// TIA Portal V19 export
FUNCTION "ALARMS" : Void   // FC10, LAD
{ S7_Optimized_Access := 'TRUE' }
// stored: SetENOAutomatically false
   VAR_TEMP   // added for the SCL form of the ladder/FBD networks
      _w1 : Bool;
   END_VAR
BEGIN

REGION Network 1: ERROR BIT
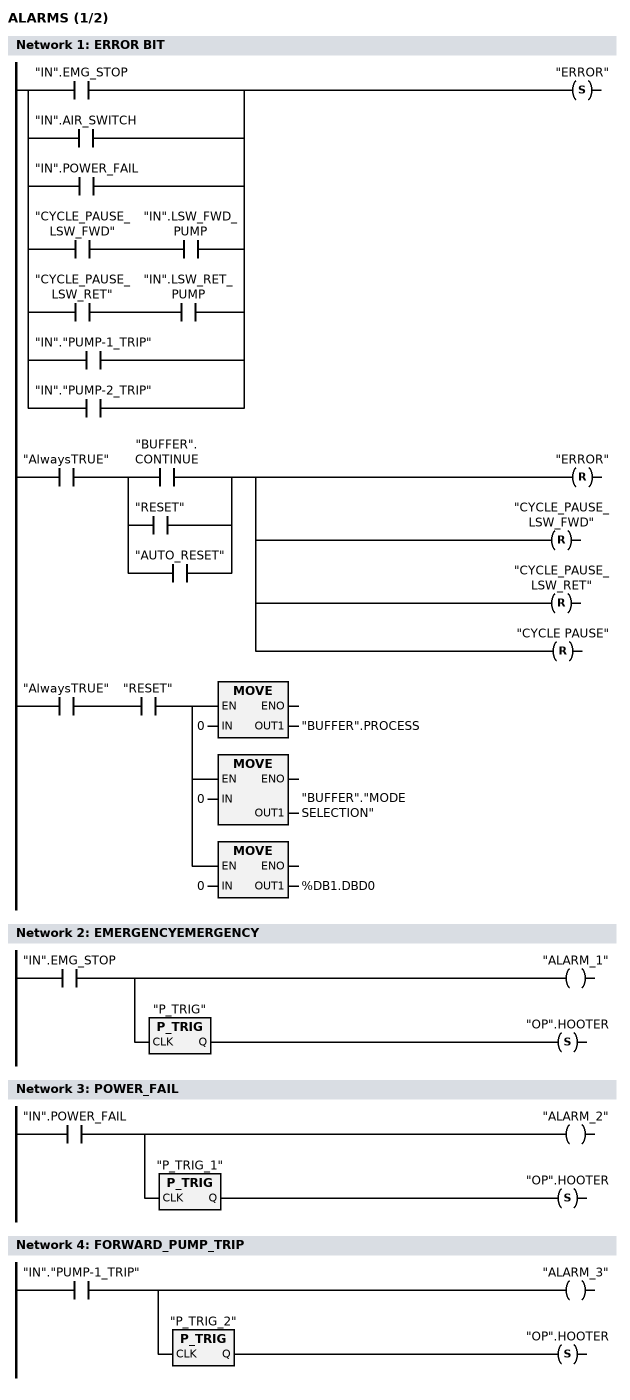
   RUNG wire#powerrail
      Contact( "IN".EMG_STOP )
      wire#w1
      S_Coil( "ERROR" )
   END_RUNG
   RUNG wire#powerrail
      Contact( "IN".AIR_SWITCH )
   END_RUNG wire#w1
   RUNG wire#powerrail
      Contact( "IN".POWER_FAIL )
   END_RUNG wire#w1
   RUNG wire#powerrail
      Contact( "CYCLE_PAUSE_LSW_FWD" )
      Contact( "IN".LSW_FWD_PUMP )
   END_RUNG wire#w1
   RUNG wire#powerrail
      Contact( "CYCLE_PAUSE_LSW_RET" )
      Contact( "IN".LSW_RET_PUMP )
   END_RUNG wire#w1
   RUNG wire#powerrail
      Contact( "IN"."PUMP-1_TRIP" )
   END_RUNG wire#w1
   RUNG wire#powerrail
      Contact( "IN"."PUMP-2_TRIP" )
   END_RUNG wire#w1
   RUNG wire#powerrail
      Contact( "AlwaysTRUE" )
      wire#w2
      Contact( "BUFFER".CONTINUE )
      wire#w3
      R_Coil( "ERROR" )
   END_RUNG
   RUNG wire#w2
      Contact( "RESET" )
   END_RUNG wire#w3
   RUNG wire#w2
      Contact( "AUTO_RESET" )
   END_RUNG wire#w3
   RUNG wire#w3
      R_Coil( "CYCLE_PAUSE_LSW_FWD" )
   END_RUNG
   RUNG wire#w3
      R_Coil( "CYCLE_PAUSE_LSW_RET" )
   END_RUNG
   RUNG wire#w3
      R_Coil( "CYCLE PAUSE" )
   END_RUNG
   RUNG wire#powerrail
      Contact( "AlwaysTRUE" )
      Contact( "RESET" )
      wire#w4
      Move(in := 0, out1 => "BUFFER".PROCESS)
   END_RUNG
   RUNG wire#w4
      Move(in := 0, out1 => "BUFFER"."MODE SELECTION")
   END_RUNG
   RUNG wire#w4
      Move(in := 0, out1 => %DB1.DBD0)
   END_RUNG
   // the same network as SCL:
   IF "IN".EMG_STOP OR "IN".AIR_SWITCH OR "IN".POWER_FAIL OR ("CYCLE_PAUSE_LSW_FWD" AND "IN".LSW_FWD_PUMP) OR ("CYCLE_PAUSE_LSW_RET" AND "IN".LSW_RET_PUMP) OR "IN"."PUMP-1_TRIP" OR "IN"."PUMP-2_TRIP" THEN
       "ERROR" := TRUE;
   END_IF;
   IF "AlwaysTRUE" AND ("BUFFER".CONTINUE OR "RESET" OR "AUTO_RESET") THEN
       "ERROR" := FALSE;
       "CYCLE_PAUSE_LSW_FWD" := FALSE;
       "CYCLE_PAUSE_LSW_RET" := FALSE;
       "CYCLE PAUSE" := FALSE;
   END_IF;
   IF "AlwaysTRUE" AND "RESET" THEN
       "BUFFER".PROCESS := 0;
       "BUFFER"."MODE SELECTION" := 0;
       %DB1.DBD0 := 0;
   END_IF;
END_REGION

REGION Network 2: EMERGENCYEMERGENCY
   RUNG wire#powerrail
      Contact( "IN".EMG_STOP )
      wire#w1
      Coil( "ALARM_1" )
   END_RUNG
   RUNG wire#w1
      P_Trig( "P_TRIG" )
      S_Coil( "OP".HOOTER )
   END_RUNG
   // the same network as SCL:
   "ALARM_1" := "IN".EMG_STOP;
   #_w1 := "IN".EMG_STOP AND NOT "P_TRIG";   // rising edge
   "P_TRIG" := "IN".EMG_STOP;
   IF #_w1 THEN "OP".HOOTER := TRUE; END_IF;
END_REGION

REGION Network 3: POWER_FAIL
   RUNG wire#powerrail
      Contact( "IN".POWER_FAIL )
      wire#w1
      Coil( "ALARM_2" )
   END_RUNG
   RUNG wire#w1
      P_Trig( "P_TRIG_1" )
      S_Coil( "OP".HOOTER )
   END_RUNG
   // the same network as SCL:
   "ALARM_2" := "IN".POWER_FAIL;
   #_w1 := "IN".POWER_FAIL AND NOT "P_TRIG_1";   // rising edge
   "P_TRIG_1" := "IN".POWER_FAIL;
   IF #_w1 THEN "OP".HOOTER := TRUE; END_IF;
END_REGION

REGION Network 4: FORWARD_PUMP_TRIP
   RUNG wire#powerrail
      Contact( "IN"."PUMP-1_TRIP" )
      wire#w1
      Coil( "ALARM_3" )
   END_RUNG
   RUNG wire#w1
      P_Trig( "P_TRIG_2" )
      S_Coil( "OP".HOOTER )
   END_RUNG
   // the same network as SCL:
   "ALARM_3" := "IN"."PUMP-1_TRIP";
   #_w1 := "IN"."PUMP-1_TRIP" AND NOT "P_TRIG_2";   // rising edge
   "P_TRIG_2" := "IN"."PUMP-1_TRIP";
   IF #_w1 THEN "OP".HOOTER := TRUE; END_IF;
END_REGION

REGION Network 5: RETURN_PUMP_TRIP
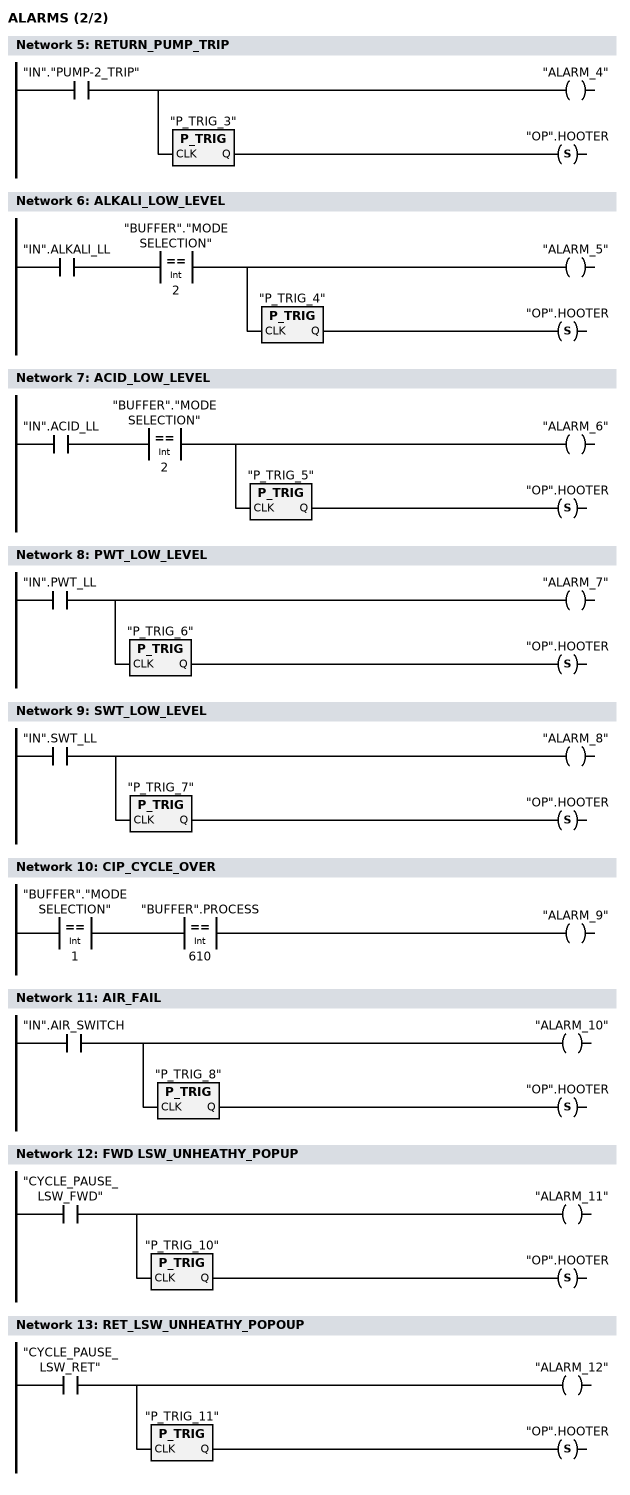
   RUNG wire#powerrail
      Contact( "IN"."PUMP-2_TRIP" )
      wire#w1
      Coil( "ALARM_4" )
   END_RUNG
   RUNG wire#w1
      P_Trig( "P_TRIG_3" )
      S_Coil( "OP".HOOTER )
   END_RUNG
   // the same network as SCL:
   "ALARM_4" := "IN"."PUMP-2_TRIP";
   #_w1 := "IN"."PUMP-2_TRIP" AND NOT "P_TRIG_3";   // rising edge
   "P_TRIG_3" := "IN"."PUMP-2_TRIP";
   IF #_w1 THEN "OP".HOOTER := TRUE; END_IF;
END_REGION

REGION Network 6: ALKALI_LOW_LEVEL
   RUNG wire#powerrail
      Contact( "IN".ALKALI_LL )
      { S7_Templates := "SrcType := Int" } EQ_Contact(in1 := "BUFFER"."MODE SELECTION", in2 := 2)
      wire#w1
      Coil( "ALARM_5" )
   END_RUNG
   RUNG wire#w1
      P_Trig( "P_TRIG_4" )
      S_Coil( "OP".HOOTER )
   END_RUNG
   // the same network as SCL:
   "ALARM_5" := "IN".ALKALI_LL AND ("BUFFER"."MODE SELECTION" = 2);
   #_w1 := "ALARM_5" AND NOT "P_TRIG_4";   // rising edge
   "P_TRIG_4" := "ALARM_5";
   IF #_w1 THEN "OP".HOOTER := TRUE; END_IF;
END_REGION

REGION Network 7: ACID_LOW_LEVEL
   RUNG wire#powerrail
      Contact( "IN".ACID_LL )
      { S7_Templates := "SrcType := Int" } EQ_Contact(in1 := "BUFFER"."MODE SELECTION", in2 := 2)
      wire#w1
      Coil( "ALARM_6" )
   END_RUNG
   RUNG wire#w1
      P_Trig( "P_TRIG_5" )
      S_Coil( "OP".HOOTER )
   END_RUNG
   // the same network as SCL:
   "ALARM_6" := "IN".ACID_LL AND ("BUFFER"."MODE SELECTION" = 2);
   #_w1 := "ALARM_6" AND NOT "P_TRIG_5";   // rising edge
   "P_TRIG_5" := "ALARM_6";
   IF #_w1 THEN "OP".HOOTER := TRUE; END_IF;
END_REGION

REGION Network 8: PWT_LOW_LEVEL
   RUNG wire#powerrail
      Contact( "IN".PWT_LL )
      wire#w1
      Coil( "ALARM_7" )
   END_RUNG
   RUNG wire#w1
      P_Trig( "P_TRIG_6" )
      S_Coil( "OP".HOOTER )
   END_RUNG
   // the same network as SCL:
   "ALARM_7" := "IN".PWT_LL;
   #_w1 := "IN".PWT_LL AND NOT "P_TRIG_6";   // rising edge
   "P_TRIG_6" := "IN".PWT_LL;
   IF #_w1 THEN "OP".HOOTER := TRUE; END_IF;
END_REGION

REGION Network 9: SWT_LOW_LEVEL
   RUNG wire#powerrail
      Contact( "IN".SWT_LL )
      wire#w1
      Coil( "ALARM_8" )
   END_RUNG
   RUNG wire#w1
      P_Trig( "P_TRIG_7" )
      S_Coil( "OP".HOOTER )
   END_RUNG
   // the same network as SCL:
   "ALARM_8" := "IN".SWT_LL;
   #_w1 := "IN".SWT_LL AND NOT "P_TRIG_7";   // rising edge
   "P_TRIG_7" := "IN".SWT_LL;
   IF #_w1 THEN "OP".HOOTER := TRUE; END_IF;
END_REGION

REGION Network 10: CIP_CYCLE_OVER
   RUNG wire#powerrail
      { S7_Templates := "SrcType := Int" } EQ_Contact(in1 := "BUFFER"."MODE SELECTION", in2 := 1)
      { S7_Templates := "SrcType := Int" } EQ_Contact(in1 := "BUFFER".PROCESS, in2 := 610)
      Coil( "ALARM_9" )
   END_RUNG
   // the same network as SCL:
   "ALARM_9" := ("BUFFER"."MODE SELECTION" = 1) AND ("BUFFER".PROCESS = 610);
END_REGION

REGION Network 11: AIR_FAIL
   RUNG wire#powerrail
      Contact( "IN".AIR_SWITCH )
      wire#w1
      Coil( "ALARM_10" )
   END_RUNG
   RUNG wire#w1
      P_Trig( "P_TRIG_8" )
      S_Coil( "OP".HOOTER )
   END_RUNG
   // the same network as SCL:
   "ALARM_10" := "IN".AIR_SWITCH;
   #_w1 := "IN".AIR_SWITCH AND NOT "P_TRIG_8";   // rising edge
   "P_TRIG_8" := "IN".AIR_SWITCH;
   IF #_w1 THEN "OP".HOOTER := TRUE; END_IF;
END_REGION

REGION Network 12: FWD LSW_UNHEATHY_POPUP
   RUNG wire#powerrail
      Contact( "CYCLE_PAUSE_LSW_FWD" )
      wire#w1
      Coil( "ALARM_11" )
   END_RUNG
   RUNG wire#w1
      P_Trig( "P_TRIG_10" )
      S_Coil( "OP".HOOTER )
   END_RUNG
   // the same network as SCL:
   "ALARM_11" := "CYCLE_PAUSE_LSW_FWD";
   #_w1 := "CYCLE_PAUSE_LSW_FWD" AND NOT "P_TRIG_10";   // rising edge
   "P_TRIG_10" := "CYCLE_PAUSE_LSW_FWD";
   IF #_w1 THEN "OP".HOOTER := TRUE; END_IF;
END_REGION

REGION Network 13: RET_LSW_UNHEATHY_POPOUP
   RUNG wire#powerrail
      Contact( "CYCLE_PAUSE_LSW_RET" )
      wire#w1
      Coil( "ALARM_12" )
   END_RUNG
   RUNG wire#w1
      P_Trig( "P_TRIG_11" )
      S_Coil( "OP".HOOTER )
   END_RUNG
   // the same network as SCL:
   "ALARM_12" := "CYCLE_PAUSE_LSW_RET";
   #_w1 := "CYCLE_PAUSE_LSW_RET" AND NOT "P_TRIG_11";   // rising edge
   "P_TRIG_11" := "CYCLE_PAUSE_LSW_RET";
   IF #_w1 THEN "OP".HOOTER := TRUE; END_IF;
END_REGION
END_FUNCTION
